# EPICS autosave request: ioc/morel/trunk/iocBoot/iocLinux/auto_positions.req
$(P)m1.DVAL
$(P)m2.DVAL
$(P)m3.DVAL
$(P)m4.DVAL
$(P)m5.DVAL
$(P)m6.DVAL
$(P)m7.DVAL
$(P)m8.DVAL

# $(P)sm1.DVAL
# $(P)sm2.DVAL
# $(P)sm3.DVAL
# $(P)sm4.DVAL
# $(P)sm5.DVAL
# $(P)sm6.DVAL
# $(P)sm7.DVAL
# $(P)sm8.DVAL
# $(P)sm9.DVAL
# $(P)sm10.DVAL
